FUNCTION func_f1: DINT
VAR_INPUT
    farg2_f1_x: DINT;
END_VAR
VAR
    farg_f1_x: DINT;
END_VAR


        farg_f1_x := farg2_f1_x;
IF ((farg_f1_x) <= (0)) THEN
    func_f1 := farg_f1_x;
    RETURN;
END_IF;
farg_f1_x := (farg_f1_x) + (1);
func_f1 := func_f2(farg_f1_x);
RETURN;

END_FUNCTION

(* stored: ProductVersion 3.1.0.18, Version 1.1.0.1 *)
